FUNCTION FUN_TimestructToTime : STRING
VAR_INPUT
	stTime : TIMESTRUCT;
END_VAR
VAR
	sTime : STRING;
END_VAR

sTime := SYSTEMTIME_TO_STRING(stTime);
FUN_TimestructToTime := RIGHT(sTime,12);

END_FUNCTION

(* stored: Version 1.1.0.1, ProductVersion 3.1.4024.9
   POU FUN_TimestructToTime: Id {796edccb-f6fd-45b7-9b19-c88a845b9034}, SpecialFunc None *)
